TYPE VTD_Settings_DUT :
STRUCT
	ID:  UINT;
	Lowest_Level:  UINT;
	Highest_Level:  UInt;
	VTD_Max_Heigh:  UInt;
	VTD_Min_Height:  UInt;
	VTD_Level_Granularity:  Int;
	Dft_Level_Offset_LE:  Int;
	Dft_Level_Offset_AE:  Int;
	Teach_Speed:  UInt;
	Creep_Speed:  UInt;
	Slow_Speed:  UInt;
	Slow_Calib_Speed:  UInt;
	Loaded_Speed:  UInt;
	Shuttle_Speed:  UInt;
	Pallet_Speed:  UInt;
	Empty_Speed:  UInt;
	Dock_speed:  UInt;
	Manual_Speed:  UInt;
	Slowdown_Count_LE:  UInt;
	Creep_Count_LE:  UInt;
	Slowdown_Count_AE:  UInt;
	Creep_Count_AE:  UInt;
	Encoder_Delta_W1:  Real;
	Encoder_Delta_W2:  Real;
	AE_Ratio:  Real;
	Encoder_Delta_Warning:  Real;
	Encoder_Delta_Error:  Real;
	Transfer_Timeout_Up:  UInt;
	Transfer_Timeout_Down:  UInt;
	Lockpins_Timeout_Extend:  UInt;
	Lockpins_Timeout_Retract:  UInt;
	Level_Detect_Timeout:  UInt;
	Teach_Timeout:  UInt;
	Chain_Slack_Timeout:  UInt;
	Level_Detect_LE:  Real;
	Acc_Range_1:  UInt;
	Acc_Range_2:  UInt;
	Acc_Range_3:  UInt;
	Weight_Range_1:  UInt;
	Weight_Range_2:  UInt;
	Weight_Range_3:  UInt;
	Teach_Values:  VTD_Levels_DUT;
END_STRUCT
END_TYPE

(* stored: Version 1.1.0.1
   DUT VTD_Settings_DUT: Id {e9c64833-e33e-4ccf-9244-2275b6dbeba0} *)
